TYPE ACRMemoryDIntEvents :
STRUCT
	_Values : ARRAY [0..GCL.cMemoryEventsMAX] OF ACRMemoryDIntEvent;
END_STRUCT
END_TYPE

(* stored: Version 1.1.0.1, ProductVersion 3.1.4020.12
   DUT ACRMemoryDIntEvents: Id {fc651e25-c8f1-4423-b0ba-ef51ef9362bd} *)
